PROGRAM MAIN
VAR
	rTemp					: REAL;
	rVar					: REAL;
	rVariablePLC			: REAL;
END_VAR

P_PLCExpert_AutoLog();
//P_PLCExpert_Independent_FBs();
//P_SQLExpert_NoDataRet();
//P_SQLExpert_DataRet();
//P_InfluxTEST();

END_PROGRAM

(* stored: Version 1.1.0.1, ProductVersion 3.1.4024.11
   POU MAIN: Id {94128c93-4a1c-4c8e-8b60-d825fdfb647f}, SpecialFunc None *)
